// TIA Portal V18 export
DATA_BLOCK "PLC8_910A3_4AO_AO_Vars"   // DB11041
{ S7_Optimized_Access := 'FALSE' }
VERSION : 0.1
// stored: AutoNumber false, DBAccessibleFromOPCUA true, IsOnlyStoredInLoadMemory false, IsWriteProtectedInAS false
   VAR
      AO1 { S7_SetPoint := 'True'} : "UDT_AOadv";   // AHU F вихід нагрівача (1.58)
      AO2 { S7_SetPoint := 'True'} : "UDT_AOadv";   // AHU F приточна/рециркуляційна заслінка (1.51/1.52)
      AO3 : "UDT_AOadv";   // Резерв
      AO4 : "UDT_AOadv";   // AHU F витяжна заслінка (1.70)
   END_VAR
BEGIN
   AO1.cFuncSystemID := 1;
   AO1.cFuncVar := 2;
   AO2.cFuncSystemID := 1;
   AO2.cFuncVar := 3;
   AO3.cFuncSystemID := 3;
   AO3.cFuncVar := 2;
   AO4.cFuncSystemID := 1;
   AO4.cFuncVar := 4;
END_DATA_BLOCK
